// TwinCAT 3 PLC project BottleFillingMachine
// ProgramVersion: 3.1.4024.0
// libraries:
//   Tc2_Standard, * (Beckhoff Automation GmbH)
//   Tc2_System, * (Beckhoff Automation GmbH)
//   Tc3_Module, * (Beckhoff Automation GmbH)
// project tree:
//   / Class Diagram.TcCD (not stored), PlcTask.TcTTO
//   DUTs/ E_AlarmState.TcDUT, E_MachineMode.TcDUT, E_MachineState.TcDUT
//   GVLs/ GVL_HMI.TcGVL
//   POUs/Conveyer/ FB_Conveyer.TcPOU, I_Conveyer.TcIO
//   POUs/ FB_MachineController.TcPOU, MAIN.TcPOU
// real-time tasks:
//   TASK PlcTask: cycle T#10ms, priority 20, ADS port 350

CONFIGURATION BottleFillingMachine
    RESOURCE PLC ON TwinCAT3
        TASK PlcTask(INTERVAL := T#10ms, PRIORITY := 20);
        PROGRAM MAIN WITH PlcTask : MAIN;
    END_RESOURCE
END_CONFIGURATION

// ---- DUTs/E_AlarmState.TcDUT
{attribute 'qualified_only'}
{attribute 'strict'}
TYPE E_AlarmState :
(
	OFF := 0,
	LEVEL_SENSOR,
	BOTTLE_SENSOR,
	CONVEYER
	
);
END_TYPE

// ---- DUTs/E_MachineMode.TcDUT
{attribute 'qualified_only'}
{attribute 'strict'}
TYPE E_MachineMode :
(
	Manual := 0,
	Auto
);
END_TYPE

// ---- DUTs/E_MachineState.TcDUT
{attribute 'qualified_only'}
{attribute 'strict'}
TYPE E_MachineState :
(
	IDLE := 0,
	WAIT_FOR_BOTTLE,
	FILLING,
	COMPLETED,
	STOPPED,
	ERROR
);
END_TYPE

// ---- GVLs/GVL_HMI.TcGVL
{attribute 'qualified_only'}
VAR_GLOBAL
	
	bStart : BOOL;
	bStop : BOOL;
	bLevelSensor : BOOL;
	bBottleSensor : BOOL;
	bReset : BOOL;
	
	bConveyerRunning : BOOL;
	bFillingValve : BOOL;
	bAlarmLamp : BOOL;
	eAlarmState : E_AlarmState;
	
	nBottleCounter : UDINT ;
	eMachineMode : E_MachineMode;
	eMachineState : E_MachineState; 
	
END_VAR

// ---- POUs/Conveyer/I_Conveyer.TcIO
INTERFACE I_Conveyer

METHOD Start : BOOL
VAR_INPUT
END_VAR
END_METHOD

METHOD Stop : BOOL
VAR_INPUT
END_VAR
END_METHOD

END_INTERFACE

// ---- POUs/MAIN.TcPOU
PROGRAM MAIN
VAR
	fbConveyer : FB_Conveyer;
	fbMachineController : FB_MachineController(_iConveyer := fbConveyer);
END_VAR


fbMachineController();

END_PROGRAM

// ---- POUs/Conveyer/FB_Conveyer.TcPOU
FUNCTION_BLOCK FB_Conveyer IMPLEMENTS I_Conveyer

VAR
END_VAR

{warning 'add method implementation '}
METHOD Start : BOOL
Start := GVL_HMI.bConveyerRunning := TRUE;
END_METHOD

{warning 'add method implementation '}
METHOD Stop : BOOL
Stop := GVL_HMI.bConveyerRunning := FALSE;
END_METHOD

END_FUNCTION_BLOCK

// ---- POUs/FB_MachineController.TcPOU
FUNCTION_BLOCK FB_MachineController
VAR
	iConveyer : I_Conveyer;
	ePreviousMachineState : E_MachineState;
	fbTimer : TON;
	tWaitTime : TIME := T#10S;
	tProcessTime : TIME := T#5S;
	fbAutoTimer : TON;
END_VAR

IF GVL_HMI.bStop THEN
	IF GVL_HMI.eMachineState =  E_MachineState.STOPPED THEN
		GVL_HMI.eMachineState := E_MachineState.IDLE;
	ELSE
		ePreviousMachineState := GVL_HMI.eMachineState ;
		GVL_HMI.eMachineState := E_MachineState.STOPPED;
	END_IF
	fbTimer(IN := FALSE, PT := tWaitTime);
	GVL_HMI.bStop := FALSE;
	
END_IF
CASE GVL_HMI.eMachineState OF
	E_MachineState.IDLE :
		IF GVL_HMI.bStart THEN
			GVL_HMI.bStart := FALSE;
			IF iConveyer <> 0 THEN
					ePreviousMachineState := GVL_HMI.eMachineState ;
					GVL_HMI.eMachineState := E_MachineState.WAIT_FOR_BOTTLE;
			ELSE
				ePreviousMachineState := GVL_HMI.eMachineState ;
				GVL_HMI.eMachineState := E_MachineState.ERROR;
			END_IF
		END_IF
		
	E_MachineState.WAIT_FOR_BOTTLE :
		iConveyer.Start();
		fbTimer ( IN:= TRUE, PT:= tWaitTime);
		IF fbTimer.Q THEN
			fbTimer(IN := FALSE);
			GVL_HMI.eAlarmState := E_AlarmState.BOTTLE_SENSOR;
			GVL_HMI.eMachineState := E_MachineState.ERROR;
		END_IF
		//AutoMode
		IF GVL_HMI.eMachineMode = E_MachineMode.Auto THEN
			fbAutoTimer(IN := TRUE, PT := tProcessTime);
			IF fbAutoTimer.Q THEN
				fbAutoTimer(IN := FALSE);
				GVL_HMI.bBottleSensor := TRUE;
			END_IF
		ELSE
			fbAutoTimer(IN := FALSE);
		END_IF
		
		IF GVL_HMI.bBottleSensor THEN
				GVL_HMI.bBottleSensor := FALSE;
				fbTimer(IN := FALSE);
				iConveyer.Stop();
				ePreviousMachineState := GVL_HMI.eMachineState ;
				GVL_HMI.eMachineState := E_MachineState.FILLING;
		END_IF
	
	E_MachineState.FILLING :
		GVL_HMI.bFillingValve := TRUE;
		fbTimer ( IN:= TRUE, PT:= tWaitTime);
		IF fbTimer.Q THEN
			fbTimer(IN := FALSE);
			GVL_HMI.eAlarmState := E_AlarmState.LEVEL_SENSOR;
			GVL_HMI.eMachineState := E_MachineState.ERROR;
		END_IF
		//AutoMode
		IF GVL_HMI.eMachineMode = E_MachineMode.Auto THEN
			fbAutoTimer(IN := TRUE, PT := tProcessTime);
			IF fbAutoTimer.Q THEN
				fbAutoTimer(IN := FALSE);
				GVL_HMI.bLevelSensor := TRUE;
			END_IF
		ELSE
			fbAutoTimer(IN := FALSE);
		END_IF
		
		IF GVL_HMI.bLevelSensor THEN
				fbTimer(IN := FALSE);
				GVL_HMI.bFillingValve := FALSE;
				ePreviousMachineState := GVL_HMI.eMachineState ;
				GVL_HMI.eMachineState := E_MachineState.COMPLETED;
		END_IF
	
	E_MachineState.COMPLETED :
			GVL_HMI.bLevelSensor := FALSE;
			iConveyer.Start();
			GVL_HMI.bBottleSensor := FALSE;
			ePreviousMachineState := GVL_HMI.eMachineState ;
			
			//Auto
			IF GVL_HMI.eMachineMode = E_MachineMode.Auto THEN
				GVL_HMI.nBottleCounter := GVL_HMI.nBottleCounter + 1;
				GVL_HMI.eMachineState := E_MachineState.WAIT_FOR_BOTTLE;
				
			ELSE
				IF GVL_HMI.bStart THEN
					GVL_HMI.nBottleCounter := GVL_HMI.nBottleCounter + 1;
					GVL_HMI.bStart := FALSE;
					GVL_HMI.eMachineState := E_MachineState.WAIT_FOR_BOTTLE;
					
				END_IF
			END_IF
			
	
	E_MachineState.STOPPED :
			iConveyer.Stop();
			GVL_HMI.bFillingValve := FALSE;
			IF GVL_HMI.bStart THEN
				GVL_HMI.bStart := FALSE;
				GVL_HMI.eMachineState := ePreviousMachineState;
			END_IF
	E_MachineState.ERROR :
		iConveyer.Stop();
		GVL_HMI.bFillingValve := FALSE;
		IF GVL_HMI.bReset THEN
			GVL_HMI.bBottleSensor := FALSE;
			GVL_HMI.bLevelSensor := FALSE;
			GVL_HMI.bReset := FALSE;
			GVL_HMI.bAlarmLamp := FALSE;
			GVL_HMI.eAlarmState := E_AlarmState.OFF;
			GVL_HMI.eMachineState := E_MachineState.IDLE;
		END_IF
END_CASE

METHOD FB_init : BOOL
VAR_INPUT
	bInitRetains : BOOL; // if TRUE, the retain variables are initialized (warm start / cold start)
	bInCopyCode : BOOL;  // if TRUE, the instance afterwards gets moved into the copy code (online change)
	_iConveyer : I_Conveyer;
END_VAR
iConveyer := _iConveyer;
END_METHOD

END_FUNCTION_BLOCK
